// TIA Portal project "Diseño estructurado" (V15.1)

(* hardware
DEVICE "S7-1200 station_1"  S7-1200 Station
   slot 0: "Rack_0"  S7-1200 Rack  Rack  V1.0
   slot 1: "PLC_1"  CPU 1214C AC/DC/Rly  6ES7 214-1BG40-0XB0  V4.2
*)

// ===== PLC "PLC_1"  CPU 1214C AC/DC/Rly =====

VAR_GLOBAL   // PLC tag table "Tabla de variables estándar"
   "Etapa0" AT %M16.0 : Bool;
   "Etapa1" AT %M16.1 : Bool;
   "Etapa2" AT %M16.2 : Bool;
   "Etapa10" AT %M100.0 : Bool;
   "Etapa11" AT %M100.1 : Bool;
   "Etapa12" AT %M100.2 : Bool;
   "Etapa20" AT %M200.0 : Bool;
   "Etapa21" AT %M200.1 : Bool;
   "Etapa22" AT %M200.2 : Bool;
   "Etapa23" AT %M200.3 : Bool;
   "Etapa24" AT %M200.4 : Bool;
   "Etapa30" AT %M300.0 : Bool;
   "Etapa31" AT %M300.1 : Bool;
   "Etapa32" AT %M300.2 : Bool;
   "Etapa33" AT %M300.3 : Bool;
   "Etapa34" AT %M300.4 : Bool;
   "Etapa35" AT %M300.5 : Bool;
   "M" AT %I1.0 : Bool;
   "A" AT %I1.1 : Bool;
   "S" AT %I1.2 : Bool;
   "TA" AT %I2.0 : Bool;
   "TB" AT %I2.1 : Bool;
   "TTAR" AT %I3.0 : Bool;
   "TTAB" AT %I3.1 : Bool;
   "PE" AT %I1.3 : Bool;
   "DI0" AT %I4.0 : Bool;
   "DI1" AT %I4.1 : Bool;
   "DI2" AT %I4.2 : Bool;
   "C1R" AT %I5.0 : Bool;
   "C2R" AT %I5.1 : Bool;
   "MT" AT %Q1.0 : Bool;
   "S1" AT %Q1.1 : Bool;
   "S2" AT %Q1.2 : Bool;
   "R1" AT %Q2.0 : Bool;
   "R2" AT %Q2.1 : Bool;
   "ROTACION_PLATO" AT %Q3.0 : Bool;
   "C1" AT %Q4.0 : Bool;
   "C2" AT %Q4.1 : Bool;
END_VAR

// folder: System blocks/Program resources

DATA_BLOCK "Temp1"   // DB1
{ S7_Optimized_Access := 'TRUE' }
AUTHOR : Simatic
FAMILY : IEC
NAME : IEC_TMR
VERSION : 1.0
// stored: InstanceOfName IEC_TIMER
"IEC_TIMER"
BEGIN
END_DATA_BLOCK

// folder: (top level)

ORGANIZATION_BLOCK "Main"   // OB1, LAD, ProgramCycle
TITLE = "Main Program Sweep (Cycle)"
{ S7_Optimized_Access := 'TRUE' }
VERSION : 0.1
   VAR_INPUT
      Initial_Call : Bool;   // Initial call of this OB
      Remanence : Bool;   // =True, if remanent data are available
   END_VAR
BEGIN

REGION Network 1
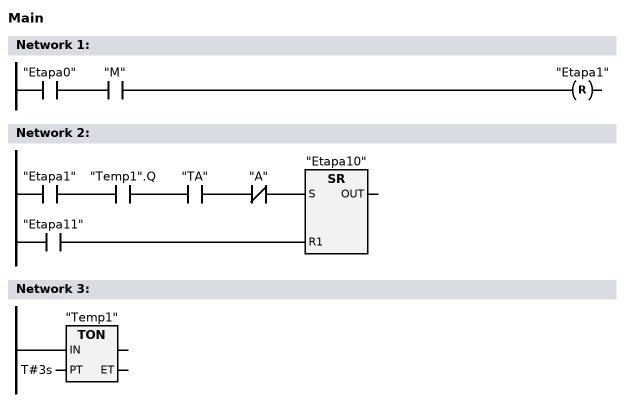
   RUNG wire#powerrail
      Contact( "Etapa0" )
      Contact( "M" )
      R_Coil( "Etapa1" )
   END_RUNG
   // the same network as SCL:
   IF "Etapa0" AND "M" THEN "Etapa1" := FALSE; END_IF;
END_REGION

REGION Network 2
   RUNG wire#powerrail
      Contact( "Etapa1" )
      Contact( "Temp1".Q )
      Contact( "TA" )
      I_Contact( "A" )
      S_SR(operand := "Etapa10", r1 := wire#w1)
   END_RUNG
   RUNG wire#powerrail
      Contact( "Etapa11" )
   END_RUNG wire#w1
   // the same network as SCL:
   IF "Etapa1" AND "Temp1".Q AND "TA" AND NOT "A" THEN
       "Etapa10" := TRUE;   // SR flip-flop
   END_IF;
   IF "Etapa11" THEN "Etapa10" := FALSE; END_IF;
END_REGION

REGION Network 3
   "Temp1".TON(IN := TRUE, PT := T#3s);
END_REGION
END_ORGANIZATION_BLOCK

ORGANIZATION_BLOCK "Startup"   // OB100, LAD, Startup
TITLE = "Complete Restart"
{ S7_Optimized_Access := 'TRUE' }
VERSION : 0.1
   VAR_INPUT
      LostRetentive : Bool;   // True if retentive data are lost
      LostRTC : Bool;   // True if date and time are lost
   END_VAR
BEGIN

REGION Network 1
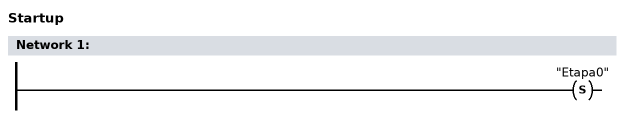
   RUNG wire#powerrail
      S_Coil( "Etapa0" )
   END_RUNG
   // the same network as SCL:
   "Etapa0" := TRUE;
END_REGION
END_ORGANIZATION_BLOCK